(* PLC project Tc2_MC2.MC_PhasingRelative Demo, tc3-libraries-kb TwinCAT 3.1 *)
(* stored: creationDateTime 2026-05-21T00:00:00, modificationDateTime 2026-05-21T00:00:00 *)

PROGRAM P_Demo_MC_PhasingRelative
  VAR
    fbAddPhase : MC_PhasingRelative;
    axisMainRoller : AXIS_REF;
    axisColorPlate : AXIS_REF;
    rtCorrectTrig : R_TRIG;
    bRunCorrection : BOOL := FALSE;
    lrPhaseErrorDeg : LREAL := 0.2;
    bCorrectionDone : BOOL;
    lrCoveredPhase : LREAL;
    nErrorID : UDINT;
  END_VAR

// =============================================================================
// 场景：套准闭环 — 视觉相机每秒反馈一个小相位偏差（如 +0.2°），用相对相位
//       调整 FB 把这个增量叠加到色版从轴上。多次调用累积修正。
// 价值：业务不用维护"当前总相位偏差"全局变量，FB 自动累加；适合做相位的
//       闭环 PID 直接输出。
// 验证：先确认主从耦合已建立（外部 MC_GearIn 已运行）；
//       bRunCorrection := TRUE 一次 → bCorrectionDone 在 ~ 0.1 s 后 TRUE，
//       lrCoveredPhase ≈ 0.2。多次触发可看到相位差累积（视觉系统反馈应回零）。
// =============================================================================

rtCorrectTrig(CLK := bRunCorrection);

fbAddPhase(
    Execute           := rtCorrectTrig.Q,
    ContinuousUpdate  := FALSE,
    PhaseShift        := lrPhaseErrorDeg,
    Velocity          := 5.0,
    Acceleration      := 50.0,
    Deceleration      := 50.0,
    Jerk              := 500.0,
    BufferMode        := MC_Aborting,
    Master            := axisMainRoller,
    Slave             := axisColorPlate,
    Done              => bCorrectionDone,
    CoveredPhaseShift => lrCoveredPhase,
    ErrorId           => nErrorID
);
END_PROGRAM
